PROGRAM MAIN
VAR
	PID_heater_enable: BOOL;  // PID Controller heater enabled ( Closed looop Control)
	PID_Servo_enable: BOOL := TRUE;   // PID Controller heater enabled ( Closed looop Control)
	pidServo  : fBDISCRETE_PID;
	pidHeater : fBDISCRETE_PID;
	States    : SeqState := SeqState.Ready;
	Cmd_Servo : R_TRIG;
	Cmd_Heater: R_TRIG;
	Cmd_ProdStart : R_TRIG;
	Cmd_ProdStop  : R_TRIG;
	HeaterON	  : BOOL;
	Rotation      : REAL;
	ToUnloadTimer : TON;
	TiMerToUnloadStart : BOOL;
	Counter : DINT;
	MoveTank : BOOL;
	StateString : STRING;
	
END_VAR

// Handling Buttons
Cmd_ProdStart(CLK:= GVL_IO.StartPr); 							// Start Process
Cmd_ProdStop(clk:=GVL_IO.StopPr);  								// Stop  Process
Cmd_Servo(clk:=MoveTank);    									// Servo Command button for testing
Cmd_Heater(clk:=GVL_IO.xPushButton2);   						// Heater Command button for testing
IF GVL_IO.Stirrer THEN     										// used to increas a counter
	Rotation := Rotation +5;									// used to rotate the stirrer in user interface
END_IF

IF Rotation = 359 THEN 											// if reached 360 degree reset
	Rotation := 0;
END_IF

ToUnloadTimer(IN := TiMerToUnloadStart ,PT := T#20S ); 			// timer to unload
// ================= START STATE SEQUENCE ======================
//
//   Your State machine program can be programmed here 
//          following an example
//

CASE States OF                       							// Sequence State ( ready, etc etc etc )
	SeqState.Ready:                  							// You can change the states if you want for your own convience
		StateString := 'Ready!';
		Counter := 0;											// sequence counter
		HeaterON := FALSE;
		IF GVL_IO.StartPr THEN 							// check if start button pressed
			States := SeqState.Fill_A;							// go to state Fill A
		END_IF
		
	SeqState.Fill_A:											// sequence state fill A
		StateString := 'Fill A';
		GVL_IO .ValveA:=TRUE;  									// open valve A				
		IF NOT GVL_IO.Level_S2 THEN 							// check if level reached s2
			GVL_IO.ValveA := FALSE;								//close valve A
			Counter := Counter + 1;									// increase counter after full cycle
			States := SeqState.Fill_B; 							// go to state Fill B
		END_IF
		
	SeqState.Fill_B:											// sequence state B
		StateString := 'Fill B';
		GVL_IO.SetPointHeater := 75; 							// set heater to 75
		HeaterON := TRUE;										//used in user interface to show heater lamp
		GVL_IO.Stirrer := TRUE; 								// set stirrer on 
		GVL_IO.ValveB := TRUE; 									// open valve B
		IF NOT GVL_IO.Level_S3 THEN 							// check if level s3 reached
			GVL_IO.ValveB := FALSE; 							// close valve B
			States := SeqState.ToUnload; 						// go to TOUnload state
		END_IF
		
	SeqState.ToUnload:											// sequence state TO Unload
		StateString := 'To Unload';
		TiMerToUnloadStart := TRUE;								// start ToUnloadTimer
		IF ToUnloadTimer.Q AND (GVL_IO.Output_Heater > 74.5 AND GVL_IO.Output_Heater < 76.5)  THEN									// if timer reached 20 sec
			TiMerToUnloadStart := FALSE;						// reset timer
			States := SeqState.MovingToDrain;					//go to MOving To drain state
		END_IF
	
	SeqState.MovingToDrain:										// sequence state moving to drain
		StateString := 'Move To Drain';
		MoveTank := TRUE;										// set move tank variable		
		GVL_IO.SetPoint_ServoX := 30;							// move tank to set point 30
		IF GVL_IO.Output_ServoX = 30 THEN						// if position reached
			MoveTank := FALSE;									// set move tank variable
			States := SeqState.Drain_1;							// go to drain 1 state
		END_IF
		
	SeqState.Drain_1:											// sequence state drain1
		StateString := 'Drain 1';
		GVL_IO.ValveC := TRUE;									//open valve c
		GVL_IO.SetPointHeater := 0;								//turn heater off
		HeaterON := FALSE;										// handle user interface variable
		IF GVL_IO.Level_S2 THEN									// if s2 level reached
			States := SeqState.Drain_2;							// go to drain 2 state
		END_IF
		
	SeqState.Drain_2:											//sequence state drain 2
		StateString := 'Drain 2';
		GVL_IO.Stirrer := FALSE;								// turn stirrer off
		IF GVL_IO.Level_S1 THEN									// if level s1 reached
			GVL_IO.ValveC := FALSE;								// close valve c 
			States := SeqState.MovingToStart;					// move to start position
		END_IF
	
	SeqState.MovingToStart: 									// sequence state move to start position
		StateString := 'Move To Start';
		MoveTank := TRUE;										// set move tank variable
		GVL_IO.SetPoint_ServoX := 0;							// set servo point to 0
		IF GVL_IO.Output_ServoX = 0 THEN						// if position 0 reached
			MoveTank := FALSE;									// set move tank variable
		IF Counter = 2 OR GVL_IO.StopPr THEN			
			States := SeqState.Ready;
		END_IF
		ELSE IF Counter < 2 AND NOT GVL_IO.StopPr THEN 
			States := SeqState.Fill_A;
		
		END_IF
		END_IF
	
		
		
		
//	
//
END_CASE
//
//

// ================ END STATE SEQUENCES=========================
// 


// =====   Executing the PID Controllers for  Position and Heater.   ===========
//==================================================================================
//
// *************  Servo with P- Controller only  **************
//
IF (MoveTank AND NOT GVL_IO.xGenCtrl_Error ) THEN
	pidServo.Setpoint:=GVL_IO.SetPoint_ServoX;  // Setpoint Servo // put in states
END_IF

pidServo.Kp:= 0.1;       //  Kp parameter
// pidServo.Ki:= xxx ; //  Ki parameter
// pidServo.Kd:= xxx ; //  Kd parameter 

pidServo.MV_max_sat:= 10;    // Maximum output PID to protect the Servo
pidServo.MV_min_sat:= -10;  // Minimum output PID    ,,     ,,
pidServo.xExt_Error:= Gvl_IO.xGenCtrl_Error;
//
pidServo.Yprocess:= LREAL_TO_REAL(GVL_IO.Output_ServoX);
//
pidServo(PID_enable:=PID_Servo_enable);  // Calling PID function Heater

// *************   Heater with P- Controller only   **********************
//
IF HeaterON THEN
   pidHeater.Setpoint:=GVL_IO.SetPointHeater;	
END_IF
IF HeaterON = FALSE THEN
	pidHeater.Setpoint := 0;
END_IF
pidHeater.Kp:= 1;         //  Kp parameter
// pidHeater.Ki:= xx ;    //  Ki parameter     
// pidHeater.Kd:= xx ;    //  Kd parameter      
pidHeater.MV_max_sat:=150;   // Maximum output PID to protect the Heater
pidHeater.MV_min_sat:= -10;  // Minimum output PID ,,     ,,
// 
pidHeater.Yprocess:=GVL_IO.Output_Heater;

pidHeater(PID_enable:= PID_heater_enable);  // Calling PID function Servo

END_PROGRAM

(* stored: Version 1.1.0.1, ProductVersion 3.1.4024.2
   POU MAIN: Id {c14fdddc-a9e2-4b2f-95bf-7a35be57990b}, SpecialFunc None *)
